FUNCTION_BLOCK ServoPosition_SetPoint

VAR CONSTANT
	nDefaultDAQ_startVal : INT := 6540;
	rDefaultEU_startVal : REAL := 3.95; //Volts
END_VAR

VAR_INPUT
	rStartValInput_EU : REAL;
	nStartValInput : INT;
END_VAR

VAR
	rStartVal_EU : REAL;
	nStartVal : INT; //El3114 DAQ resolution, 16 bit (1 bit = sign bit)
END_VAR
VAR // added by the converter: edge detectors and wires of the graphical bodies
    _w1, _w2 : BOOL;
END_VAR

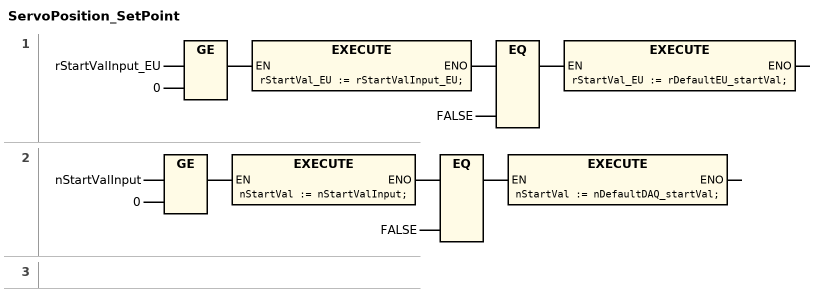
// NETWORK 1
_w1 := rStartValInput_EU >= 0;
IF _w1 THEN rStartVal_EU := rStartValInput_EU; END_IF
IF _w1 = FALSE THEN rStartVal_EU := rDefaultEU_startVal; END_IF

// NETWORK 2
_w2 := nStartValInput >= 0;
IF _w2 THEN nStartVal := nStartValInput; END_IF
IF _w2 = FALSE THEN nStartVal := nDefaultDAQ_startVal; END_IF

// NETWORK 3

METHOD PercentPosition : REAL

VAR
	rDAQtomA_ConvFac : REAL; //DAQ signed 16 bit number to EU (mA)
	rmAToPercent : REAL; //Conversion factor from mA to %
END_VAR
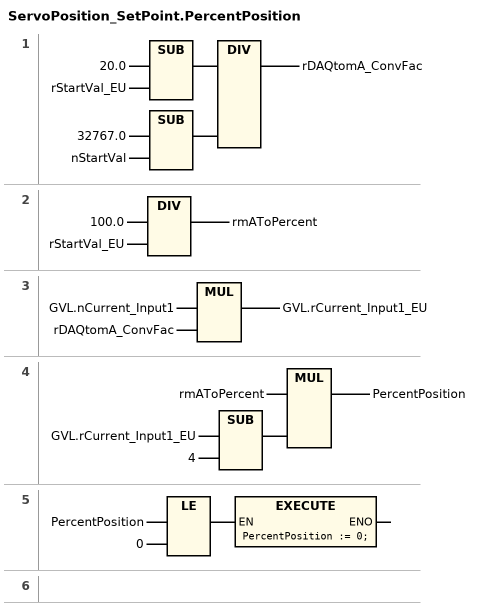
// NETWORK 1
rDAQtomA_ConvFac := (20.0 - rStartVal_EU) / (32767.0 - nStartVal);

// NETWORK 2
rmAToPercent := 100.0 / rStartVal_EU;

// NETWORK 3
GVL.rCurrent_Input1_EU := GVL.nCurrent_Input1 * rDAQtomA_ConvFac;

// NETWORK 4
PercentPosition := rmAToPercent * (GVL.rCurrent_Input1_EU - 4);

// NETWORK 5
IF PercentPosition <= 0 THEN PercentPosition := 0; END_IF

// NETWORK 6
END_METHOD

END_FUNCTION_BLOCK

(* stored: Version 1.1.0.1, ProductVersion 3.1.4024.12
   POU ServoPosition_SetPoint: Id {b8b83adc-b271-4dd1-a911-513782680edf}, SpecialFunc None
   Method PercentPosition: Id {d4806622-a0c7-46ed-a1d9-640951d0c6ba} *)
